(* Logix 5000 project; controller p65 vendor 1 type 14 code 85 rev 20.11; software revision 20.01; part 3 of 7 *)
(* tags used below, declared in another part *)
   BatterycanSupplyPower : ALIAS FOR DINT00_22.0;
   Batterycharge : ALIAS FOR REAL00_3;
   BatteryreqDischarge : ALIAS FOR DINT00_22.30;
   BatteryreqDisconnect : ALIAS FOR DINT00_22.31;
   CommreqConnect : ALIAS FOR DINT00_27.16;
   CommreqDisconnect : ALIAS FOR DINT00_27.17;
   DCMicroGridcanNotifyUser : ALIAS FOR DINT00_23.5;
   DCMicroGridinitialPowerRate : ALIAS FOR REAL00_29;
   DCMicroGridisInOperation : ALIAS FOR DINT00_23.8;
   DCMicroGridisShutdown : ALIAS FOR DINT00_23.9;
   DCMicroGridisSimulating : ALIAS FOR DINT00_23.10;
   DCMicroGridisStarted : ALIAS FOR DINT00_23.11;
   DCMicroGridlowestSupportedPriority : ALIAS FOR DINT00_17;
   DCMicroGridmaxPowerRate : ALIAS FOR REAL00_185;
   DCMicroGridmorePowerAvailable : ALIAS FOR DINT00_32.12;
   DCMicroGridnotificationTimer : ALIAS FOR CLTIMER00_94;
   DCMicroGridpowerRate : ALIAS FOR REAL00_186;
   DCMicroGridpowerRateIncrement : REAL;
   DCMicroGridrecruitingPhase : ALIAS FOR DINT00_18;
   DCMicroGridreqReset : ALIAS FOR DINT00_32.13;
   DCMicroGridreqShutdown : ALIAS FOR DINT00_32.14;
   DCMicroGridreqStartup : ALIAS FOR DINT00_32.15;
   DCMicroGridResetEventFail : ALIAS FOR DINT00_32.16;
   DCMicroGridResetEventSuccess : ALIAS FOR DINT00_32.17;
   DCMicroGridResetFailTimer : ALIAS FOR CLTIMER00_95;
   DCMicroGridResetInProcess : ALIAS FOR DINT00_32.18;
   DCMicroGridResetMsg : ALIAS FOR MESSAGE00_25;
   DCMicroGridResetSuccessTimer : ALIAS FOR CLTIMER00_96;
   DCMicroGridShutdownEventFail : ALIAS FOR DINT00_32.19;
   DCMicroGridShutdownEventSuccess : ALIAS FOR DINT00_32.20;
   DCMicroGridShutdownFailTimer : ALIAS FOR CLTIMER00_97;
   DCMicroGridShutdownInProcess : ALIAS FOR DINT00_32.21;
   DCMicroGridShutdownMsg : ALIAS FOR MESSAGE00_26;
   DCMicroGridShutdownSuccessTimer : ALIAS FOR CLTIMER00_98;
   DCMicroGridsourcesProvidingExcessPower : ALIAS FOR DINT00_33.7;
   DCMicroGridStartupEventFail : ALIAS FOR DINT00_33.8;
   DCMicroGridStartupEventSuccess : ALIAS FOR DINT00_33.9;
   DCMicroGridStartupFailTimer : ALIAS FOR CLTIMER00_100;
   DCMicroGridStartupInProcess : ALIAS FOR DINT00_33.10;
   DCMicroGridStartupMsg : ALIAS FOR MESSAGE00_27;
   DCMicroGridStartupSuccessTimer : ALIAS FOR CLTIMER00_101;
   DCMicroGridtest : ALIAS FOR REAL00_192;
   DCMicroGridtestout : ALIAS FOR REAL00_193;
   DCMicroGriduserNotified : ALIAS FOR DINT00_33.11;
   House01accountBalance : ALIAS FOR REAL00_115;
   House01accountDepositRate : ALIAS FOR REAL00_116;
   House01Bclose : ALIAS FOR Local:3:O.Data.0;
   House01BcloseHILS : ALIAS FOR plc1_local_6[0].0;
   House01BcloseProxy : ALIAS FOR DINT00_28.9;
   House01BintReqClose : ALIAS FOR DINT00_28.10;
   House01BisClosed : ALIAS FOR DINT00_28.11;
   House01BisOpen : ALIAS FOR DINT00_28.12;
   House01BreqClose : ALIAS FOR DINT00_28.13;
   House01BreqOpen : ALIAS FOR DINT00_28.14;
   House01commandChanged : ALIAS FOR DINT00_28.15;
   House01commandChangedTimer : ALIAS FOR CLTIMER00_50;
   House01current : ALIAS FOR REAL00_117;
   House01currentHILS : ALIAS FOR plc1_local_2[0];
   House01currentRaw : ALIAS FOR Local:1:I.Ch12Data;
   House01deadband : ALIAS FOR REAL00_118;
   House01depositTimer : ALIAS FOR CLTIMER00_51;
   House01DisconnectPowerEventFail : ALIAS FOR DINT00_28.16;
   House01DisconnectPowerEventSuccess : ALIAS FOR DINT00_28.17;
   House01DisconnectPowerFailTimer : ALIAS FOR CLTIMER00_52;
   House01DisconnectPowerInProcess : ALIAS FOR DINT00_28.18;
   House01DisconnectPowerMsg : ALIAS FOR MESSAGE00_12;
   House01DisconnectPowerSuccessTimer : ALIAS FOR CLTIMER00_53;
   House01failedToConnect : ALIAS FOR DINT00_28.19;
   House01failedToDisconnect : ALIAS FOR DINT00_28.20;
   House01fundsAvailable : ALIAS FOR DINT00_28.21;
   House01incrementToAdd : ALIAS FOR REAL00_119;
   House01incrementToSubtract : ALIAS FOR REAL00_120;
   House01initialAccountBalance : ALIAS FOR REAL00_121;
   House01intReqConnect : ALIAS FOR DINT00_28.22;
   House01isConnected : ALIAS FOR DINT00_28.23;
   House01isDisconnected : ALIAS FOR DINT00_28.24;
   House01minBalance : ALIAS FOR REAL00_122;
   House01minBalanceToReconnect : ALIAS FOR REAL00_123;
   House01minTime : ALIAS FOR REAL00_124;
   House01powerRate : ALIAS FOR REAL00_125;
   House01powerRateMax : REAL;
   House01priority : ALIAS FOR DINT00_12;
   House01PurchasePowerEventFail : ALIAS FOR DINT00_28.25;
   House01PurchasePowerEventSuccess : ALIAS FOR DINT00_28.26;
   House01PurchasePowerFailTimer : ALIAS FOR CLTIMER00_54;
   House01PurchasePowerInProcess : ALIAS FOR DINT00_28.27;
   House01PurchasePowerMsg : ALIAS FOR MESSAGE00_13;
   House01PurchasePowerSuccessTimer : ALIAS FOR CLTIMER00_55;
   House01reqConnect : ALIAS FOR DINT00_28.28;
   House01reqDisconnect : ALIAS FOR DINT00_28.29;
   House01runningOut : ALIAS FOR DINT00_28.30;
   House01spendingRate : ALIAS FOR REAL00_126;
   House01timeRemaining : ALIAS FOR REAL00_127;
   House01usageTimer : ALIAS FOR CLTIMER00_56;
   House02accountBalance : ALIAS FOR REAL00_128;
   House02initialAccountBalance : ALIAS FOR REAL00_134;
   House02powerRate : ALIAS FOR REAL00_138;
   House02powerRateMax : REAL;
   House02priority : ALIAS FOR DINT00_13;
   House02reqConnect : ALIAS FOR DINT00_29.18;
   House02reqDisconnect : ALIAS FOR DINT00_29.19;
   House03accountBalance : ALIAS FOR REAL00_141;
   House03initialAccountBalance : ALIAS FOR REAL00_147;
   House03powerRate : ALIAS FOR REAL00_151;
   House03powerRateMax : REAL;
   House03priority : ALIAS FOR DINT00_14;
   House03reqConnect : ALIAS FOR DINT00_30.8;
   House03reqDisconnect : ALIAS FOR DINT00_30.9;
   House04accountBalance : ALIAS FOR REAL00_154;
   House04initialAccountBalance : ALIAS FOR REAL00_160;
   House04powerRate : ALIAS FOR REAL00_164;
   House04powerRateMax : REAL;
   House04priority : ALIAS FOR DINT00_15;
   House04reqConnect : ALIAS FOR DINT00_30.30;
   House04reqDisconnect : ALIAS FOR DINT00_30.31;
   House05accountBalance : ALIAS FOR REAL00_167;
   House05initialAccountBalance : ALIAS FOR REAL00_173;
   House05powerRate : ALIAS FOR REAL00_177;
   House05powerRateMax : REAL;
   House05priority : ALIAS FOR DINT00_16;
   House05reqConnect : ALIAS FOR DINT00_31.20;
   House05reqDisconnect : ALIAS FOR DINT00_31.21;
   Load01accountBalance : ALIAS FOR REAL00_37;
   Load01initialAccountBalance : ALIAS FOR REAL00_43;
   Load01powerRate : ALIAS FOR REAL00_47;
   Load01powerRateMax : REAL;
   Load01priority : ALIAS FOR DINT00_5;
   Load01reqConnect : ALIAS FOR DINT00_24.18;
   Load01reqDisconnect : ALIAS FOR DINT00_24.19;
   Load02accountBalance : ALIAS FOR REAL00_50;
   Load02initialAccountBalance : ALIAS FOR REAL00_56;
   Load02powerRate : ALIAS FOR REAL00_60;
   Load02powerRateMax : REAL;
   Load02priority : ALIAS FOR DINT00_6;
   Load02reqConnect : ALIAS FOR DINT00_25.8;
   Load02reqDisconnect : ALIAS FOR DINT00_25.9;
   Load03accountBalance : ALIAS FOR REAL00_63;
   Load03initialAccountBalance : ALIAS FOR REAL00_69;
   Load03powerRate : ALIAS FOR REAL00_73;
   Load03powerRateMax : REAL;
   Load03priority : ALIAS FOR DINT00_7;
   Load03reqConnect : ALIAS FOR DINT00_25.30;
   Load03reqDisconnect : ALIAS FOR DINT00_25.31;
   Load04accountBalance : ALIAS FOR REAL00_76;
   Load04initialAccountBalance : ALIAS FOR REAL00_82;
   Load04powerRate : ALIAS FOR REAL00_86;
   Load04powerRateMax : REAL;
   Load04priority : ALIAS FOR DINT00_8;
   Load04reqConnect : ALIAS FOR DINT00_26.20;
   Load04reqDisconnect : ALIAS FOR DINT00_26.21;
   Load05accountBalance : ALIAS FOR REAL00_89;
   Load05initialAccountBalance : ALIAS FOR REAL00_95;
   Load05powerRate : ALIAS FOR REAL00_99;
   Load05powerRateMax : REAL;
   Load05priority : ALIAS FOR DINT00_9;
   Load05reqConnect : ALIAS FOR DINT00_27.10;
   Load05reqDisconnect : ALIAS FOR DINT00_27.11;
   LoadslowVoltage : ALIAS FOR DINT00_27.23;
   PricedecreaseInProcess : BOOL;
   PriceDecreaseTimer : TIMER;
   PriceIncreaseTimer : TIMER;
   PriorityDecreaseInProcess : BOOL;
   PriorityDecreaseTimer : TIMER;
   PriorityIncreaseTimer : TIMER;
   ResreqConnect : ALIAS FOR DINT00_31.29;
   ResreqDisconnect : ALIAS FOR DINT00_31.30;
   SolarPanelcanSupplyPower : ALIAS FOR DINT00_32.28;
   SolarPanelprovidingExcessPower : ALIAS FOR DINT00_33.4;
   SolarPanelreqConnect : ALIAS FOR DINT00_33.5;
   SolarPanelreqDisconnect : ALIAS FOR DINT00_33.6;
   UsingAgents : BOOL;

PROGRAM DCMicroGrid   (* main routine DCMicroGrid *)

ROUTINE DCMicroGrid   (* ladder *)
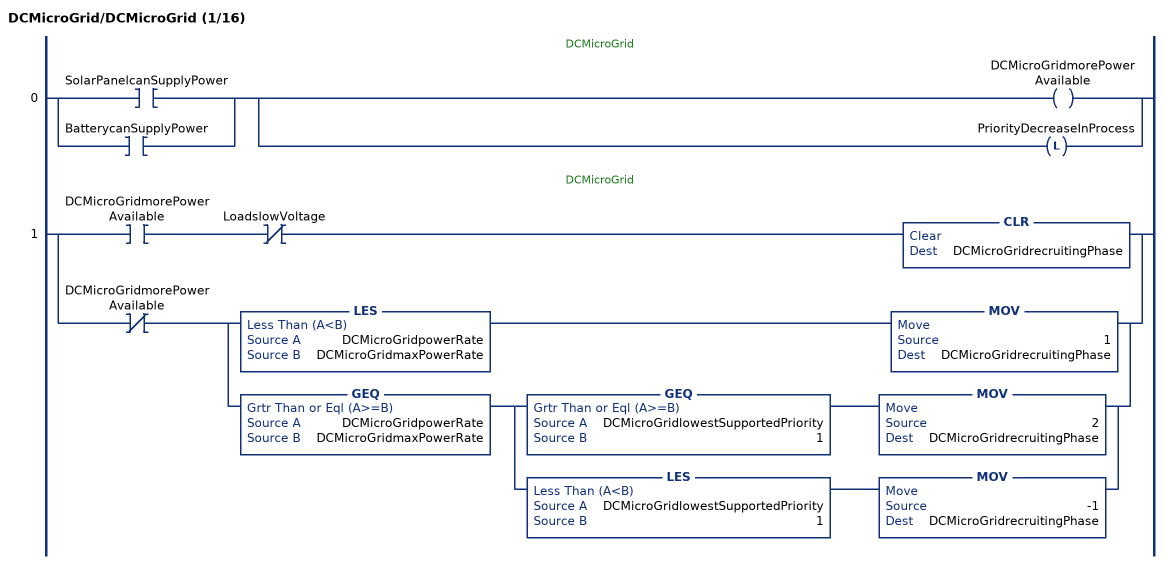
   // DCMicroGrid
   0: [XIC(SolarPanelcanSupplyPower) ,XIC(BatterycanSupplyPower) ][OTE(DCMicroGridmorePowerAvailable) ,OTL(PriorityDecreaseInProcess) ];
   // DCMicroGrid
   1: [XIC(DCMicroGridmorePowerAvailable) XIO(LoadslowVoltage) CLR(DCMicroGridrecruitingPhase) ,XIO(DCMicroGridmorePowerAvailable) [LES(DCMicroGridpowerRate,DCMicroGridmaxPowerRate) MOV(1,DCMicroGridrecruitingPhase) ,GEQ(DCMicroGridpowerRate,DCMicroGridmaxPowerRate) [GEQ(DCMicroGridlowestSupportedPriority,1) MOV(2,DCMicroGridrecruitingPhase) ,LES(DCMicroGridlowestSupportedPriority,1) MOV(-1,DCMicroGridrecruitingPhase) ] ] ];
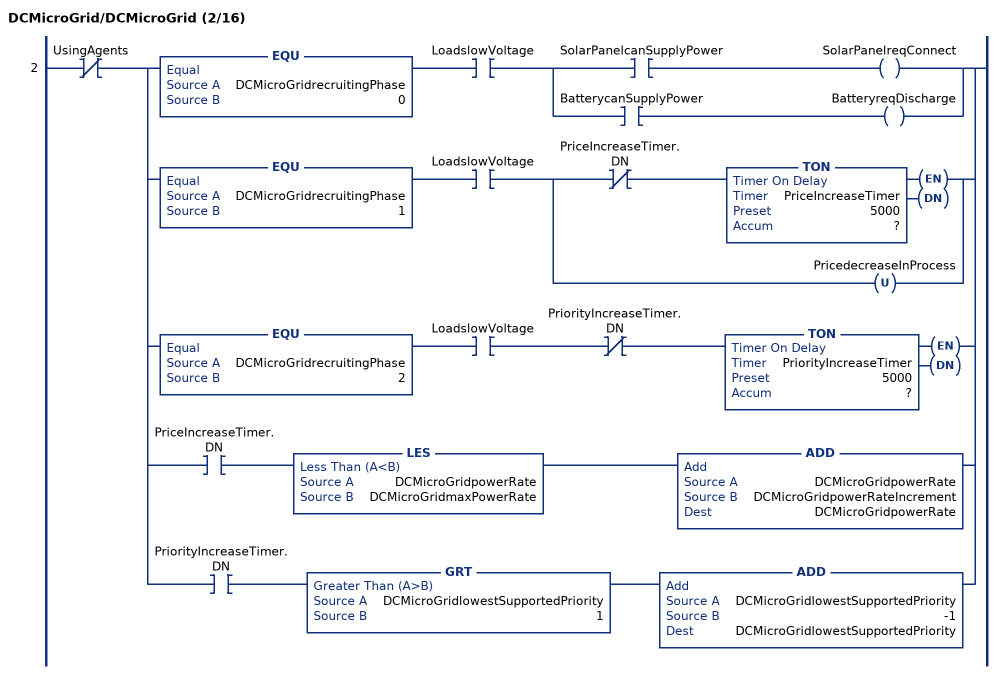
   2: XIO(UsingAgents)[EQU(DCMicroGridrecruitingPhase,0) XIC(LoadslowVoltage) [XIC(SolarPanelcanSupplyPower) OTE(SolarPanelreqConnect) ,XIC(BatterycanSupplyPower) OTE(BatteryreqDischarge) ] ,EQU(DCMicroGridrecruitingPhase,1) XIC(LoadslowVoltage) [XIO(PriceIncreaseTimer.DN) TON(PriceIncreaseTimer,?,?) ,OTU(PricedecreaseInProcess) ] ,EQU(DCMicroGridrecruitingPhase,2) XIC(LoadslowVoltage) XIO(PriorityIncreaseTimer.DN) TON(PriorityIncreaseTimer,?,?) ,XIC(PriceIncreaseTimer.DN) LES(DCMicroGridpowerRate,DCMicroGridmaxPowerRate) ADD(DCMicroGridpowerRate,DCMicroGridpowerRateIncrement,DCMicroGridpowerRate) ,XIC(PriorityIncreaseTimer.DN) GRT(DCMicroGridlowestSupportedPriority,1) ADD(DCMicroGridlowestSupportedPriority,-1,DCMicroGridlowestSupportedPriority) ];
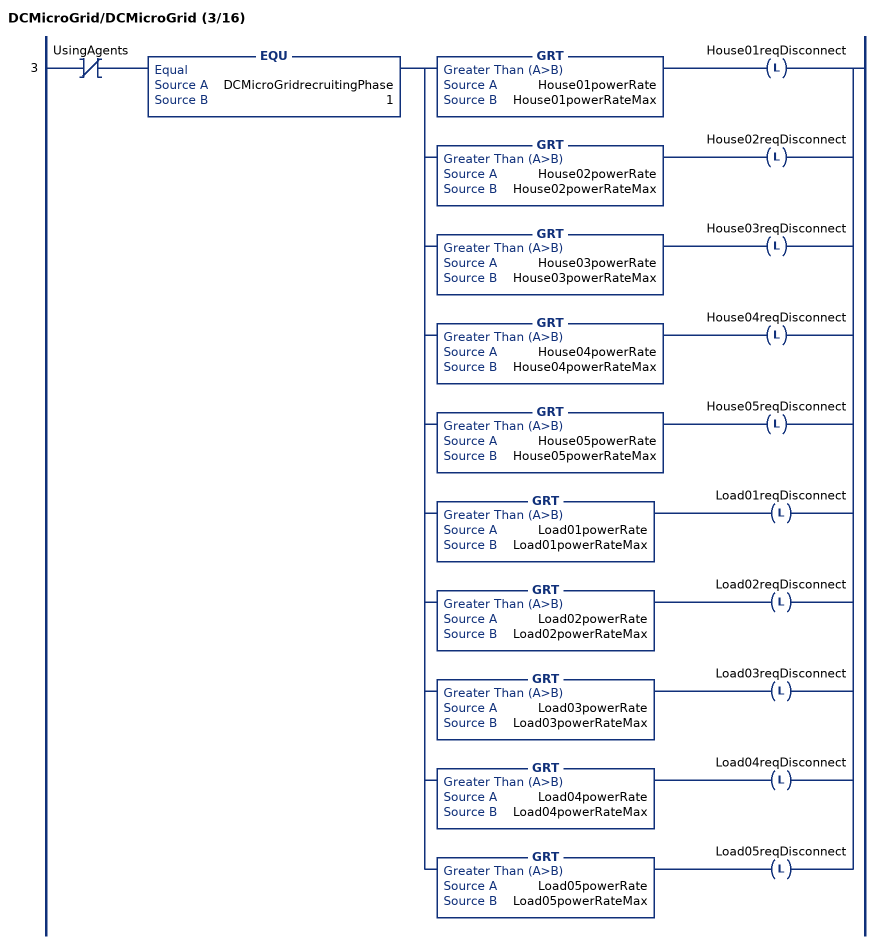
   3: XIO(UsingAgents)EQU(DCMicroGridrecruitingPhase,1)[GRT(House01powerRate,House01powerRateMax) OTL(House01reqDisconnect) ,GRT(House02powerRate,House02powerRateMax) OTL(House02reqDisconnect) ,GRT(House03powerRate,House03powerRateMax) OTL(House03reqDisconnect) ,GRT(House04powerRate,House04powerRateMax) OTL(House04reqDisconnect) ,GRT(House05powerRate,House05powerRateMax) OTL(House05reqDisconnect) ,GRT(Load01powerRate,Load01powerRateMax) OTL(Load01reqDisconnect) ,GRT(Load02powerRate,Load02powerRateMax) OTL(Load02reqDisconnect) ,GRT(Load03powerRate,Load03powerRateMax) OTL(Load03reqDisconnect) ,GRT(Load04powerRate,Load04powerRateMax) OTL(Load04reqDisconnect) ,GRT(Load05powerRate,Load05powerRateMax) OTL(Load05reqDisconnect) ];
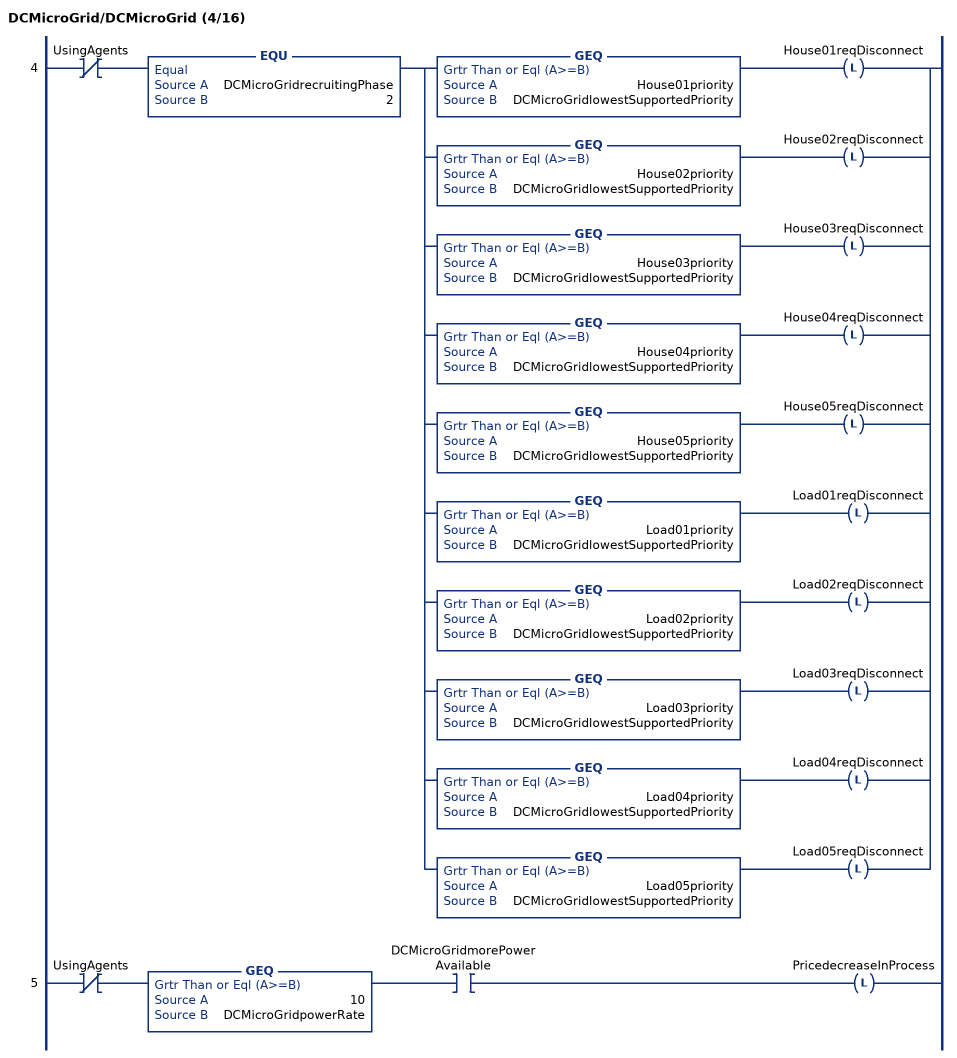
   4: XIO(UsingAgents)EQU(DCMicroGridrecruitingPhase,2)[GEQ(House01priority,DCMicroGridlowestSupportedPriority) OTL(House01reqDisconnect) ,GEQ(House02priority,DCMicroGridlowestSupportedPriority) OTL(House02reqDisconnect) ,GEQ(House03priority,DCMicroGridlowestSupportedPriority) OTL(House03reqDisconnect) ,GEQ(House04priority,DCMicroGridlowestSupportedPriority) OTL(House04reqDisconnect) ,GEQ(House05priority,DCMicroGridlowestSupportedPriority) OTL(House05reqDisconnect) ,GEQ(Load01priority,DCMicroGridlowestSupportedPriority) OTL(Load01reqDisconnect) ,GEQ(Load02priority,DCMicroGridlowestSupportedPriority) OTL(Load02reqDisconnect) ,GEQ(Load03priority,DCMicroGridlowestSupportedPriority) OTL(Load03reqDisconnect) ,GEQ(Load04priority,DCMicroGridlowestSupportedPriority) OTL(Load04reqDisconnect) ,GEQ(Load05priority,DCMicroGridlowestSupportedPriority) OTL(Load05reqDisconnect) ];
   5: XIO(UsingAgents)GEQ(10,DCMicroGridpowerRate)XIC(DCMicroGridmorePowerAvailable)OTL(PricedecreaseInProcess);
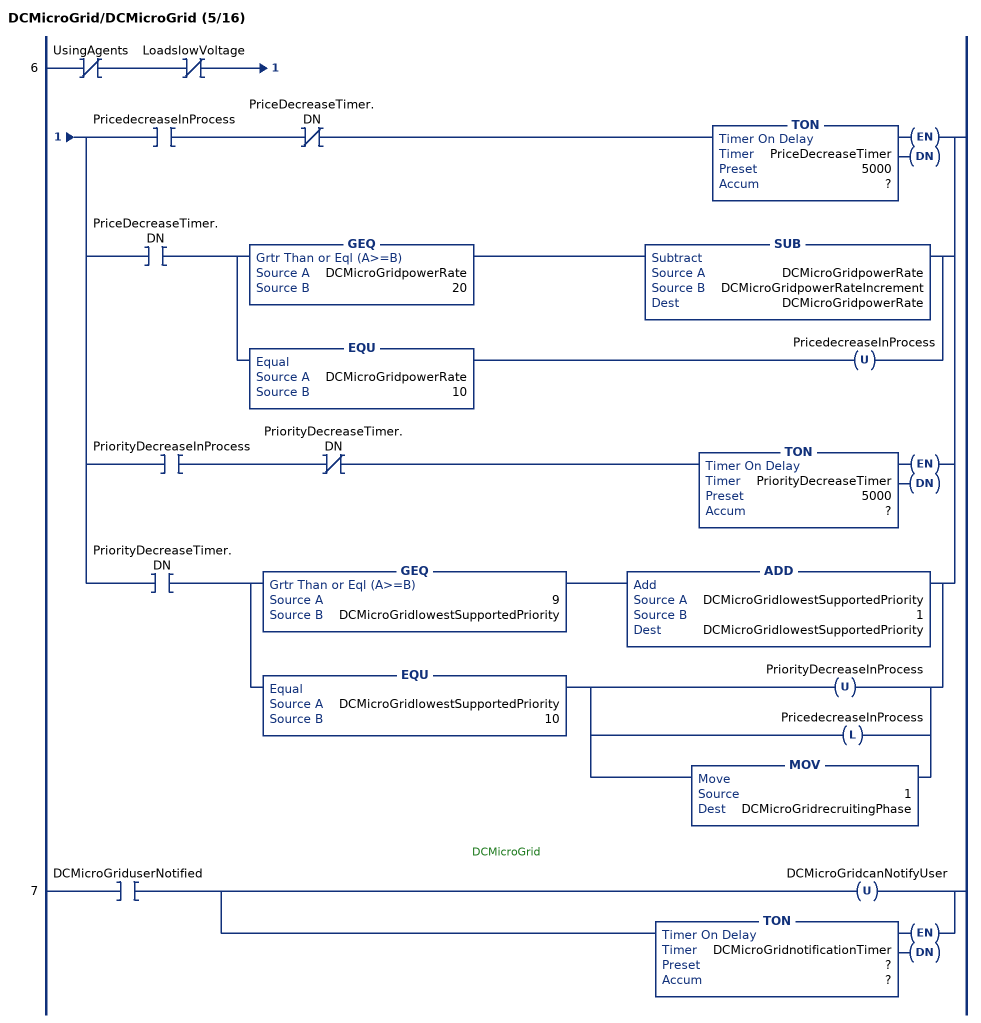
   6: XIO(UsingAgents)XIO(LoadslowVoltage)[XIC(PricedecreaseInProcess) XIO(PriceDecreaseTimer.DN) TON(PriceDecreaseTimer,?,?) ,XIC(PriceDecreaseTimer.DN) [GEQ(DCMicroGridpowerRate,20) SUB(DCMicroGridpowerRate,DCMicroGridpowerRateIncrement,DCMicroGridpowerRate) ,EQU(DCMicroGridpowerRate,10) OTU(PricedecreaseInProcess) ] ,XIC(PriorityDecreaseInProcess) XIO(PriorityDecreaseTimer.DN) TON(PriorityDecreaseTimer,?,?) ,XIC(PriorityDecreaseTimer.DN) [GEQ(9,DCMicroGridlowestSupportedPriority) ADD(DCMicroGridlowestSupportedPriority,1,DCMicroGridlowestSupportedPriority) ,EQU(DCMicroGridlowestSupportedPriority,10) [OTU(PriorityDecreaseInProcess) ,OTL(PricedecreaseInProcess) ,MOV(1,DCMicroGridrecruitingPhase) ] ] ];
   // DCMicroGrid
   7: XIC(DCMicroGriduserNotified)[OTU(DCMicroGridcanNotifyUser) ,TON(DCMicroGridnotificationTimer,?,?) ];
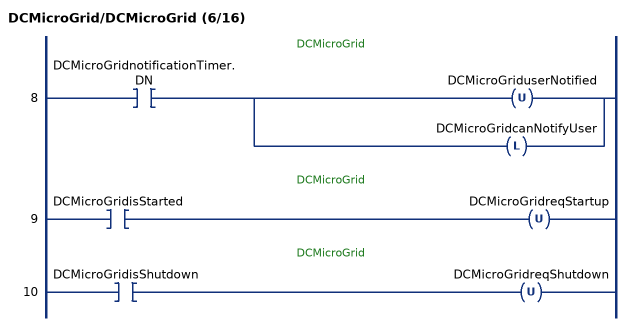
   // DCMicroGrid
   8: XIC(DCMicroGridnotificationTimer.DN)[OTU(DCMicroGriduserNotified) ,OTL(DCMicroGridcanNotifyUser) ];
   // DCMicroGrid
   9: XIC(DCMicroGridisStarted)OTU(DCMicroGridreqStartup);
   // DCMicroGrid
   10: XIC(DCMicroGridisShutdown)OTU(DCMicroGridreqShutdown);
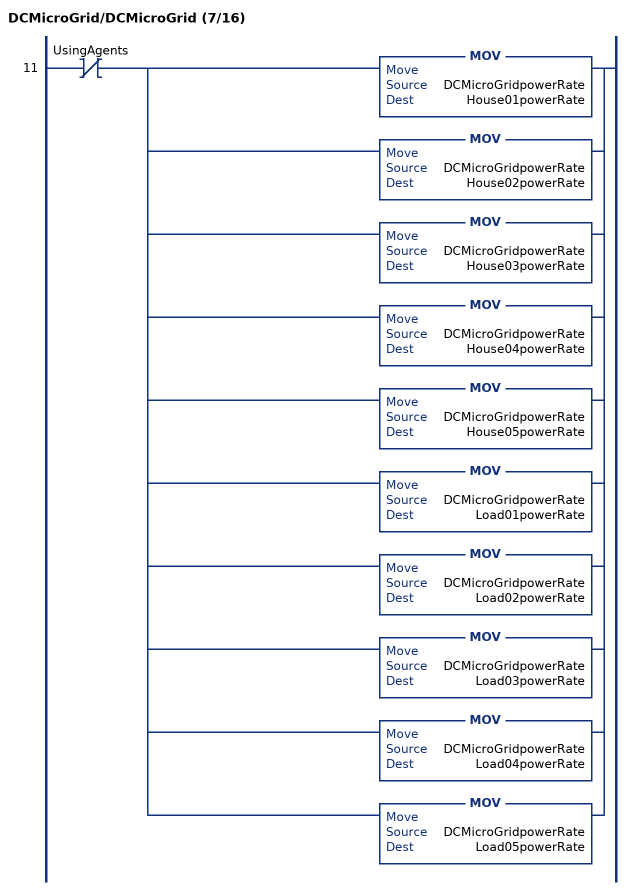
   11: XIO(UsingAgents)[MOV(DCMicroGridpowerRate,House01powerRate) ,MOV(DCMicroGridpowerRate,House02powerRate) ,MOV(DCMicroGridpowerRate,House03powerRate) ,MOV(DCMicroGridpowerRate,House04powerRate) ,MOV(DCMicroGridpowerRate,House05powerRate) ,MOV(DCMicroGridpowerRate,Load01powerRate) ,MOV(DCMicroGridpowerRate,Load02powerRate) ,MOV(DCMicroGridpowerRate,Load03powerRate) ,MOV(DCMicroGridpowerRate,Load04powerRate) ,MOV(DCMicroGridpowerRate,Load05powerRate) ];
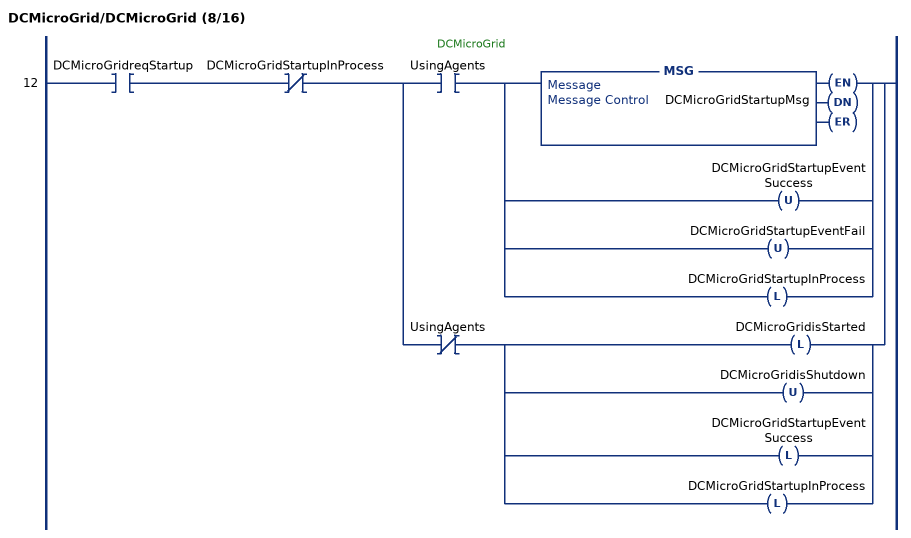
   // DCMicroGrid
   12: XIC(DCMicroGridreqStartup)XIO(DCMicroGridStartupInProcess)[XIC(UsingAgents) [MSG(DCMicroGridStartupMsg) ,OTU(DCMicroGridStartupEventSuccess) ,OTU(DCMicroGridStartupEventFail) ,OTL(DCMicroGridStartupInProcess) ] ,XIO(UsingAgents) [OTL(DCMicroGridisStarted) ,OTU(DCMicroGridisShutdown) ,OTL(DCMicroGridStartupEventSuccess) ,OTL(DCMicroGridStartupInProcess) ] ];
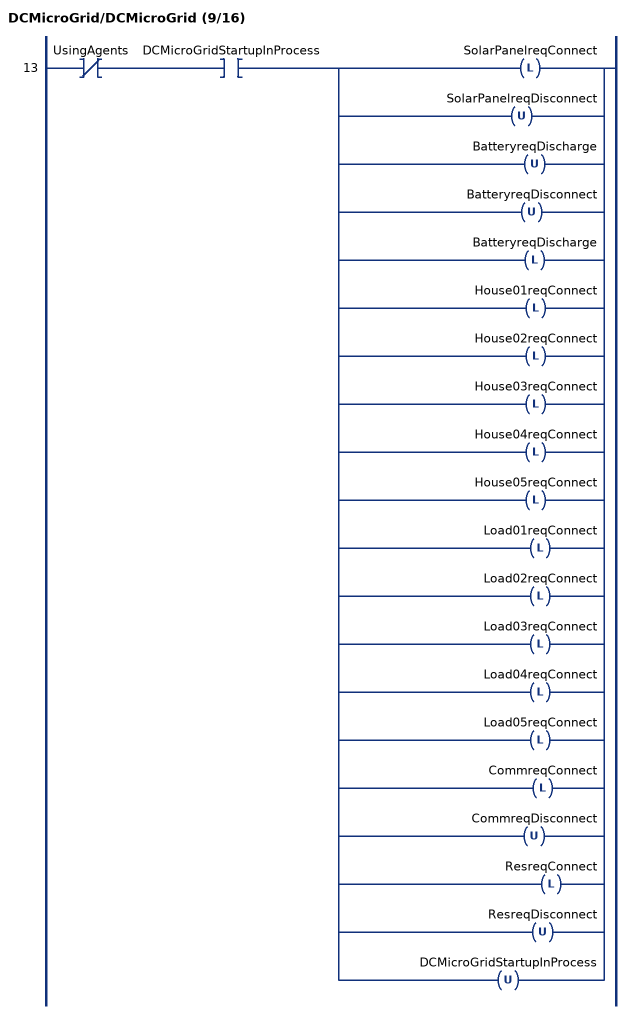
   13: XIO(UsingAgents)XIC(DCMicroGridStartupInProcess)[OTL(SolarPanelreqConnect) ,OTU(SolarPanelreqDisconnect) ,OTU(BatteryreqDischarge) ,OTU(BatteryreqDisconnect) ,OTL(BatteryreqDischarge) ,OTL(House01reqConnect) ,OTL(House02reqConnect) ,OTL(House03reqConnect) ,OTL(House04reqConnect) ,OTL(House05reqConnect) ,OTL(Load01reqConnect) ,OTL(Load02reqConnect) ,OTL(Load03reqConnect) ,OTL(Load04reqConnect) ,OTL(Load05reqConnect) ,OTL(CommreqConnect) ,OTU(CommreqDisconnect) ,OTL(ResreqConnect) ,OTU(ResreqDisconnect) ,OTU(DCMicroGridStartupInProcess) ];
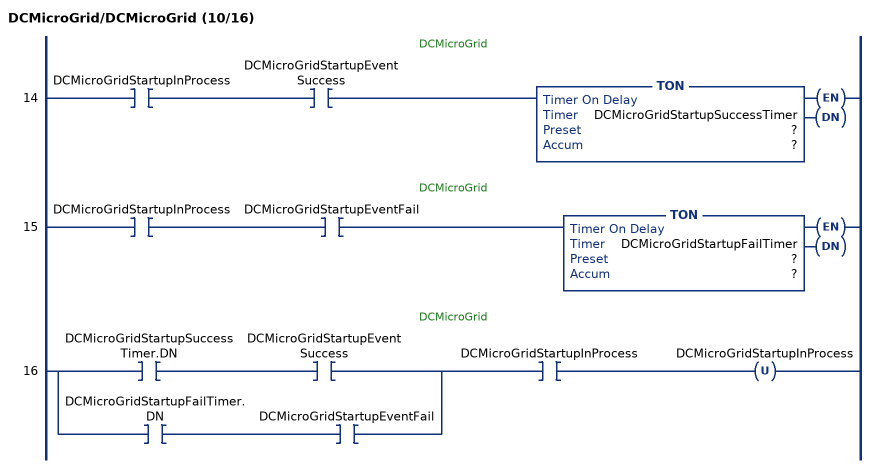
   // DCMicroGrid
   14: XIC(DCMicroGridStartupInProcess)XIC(DCMicroGridStartupEventSuccess)TON(DCMicroGridStartupSuccessTimer,?,?);
   // DCMicroGrid
   15: XIC(DCMicroGridStartupInProcess)XIC(DCMicroGridStartupEventFail)TON(DCMicroGridStartupFailTimer,?,?);
   // DCMicroGrid
   16: [XIC(DCMicroGridStartupSuccessTimer.DN) XIC(DCMicroGridStartupEventSuccess) ,XIC(DCMicroGridStartupFailTimer.DN) XIC(DCMicroGridStartupEventFail) ]XIC(DCMicroGridStartupInProcess)OTU(DCMicroGridStartupInProcess);
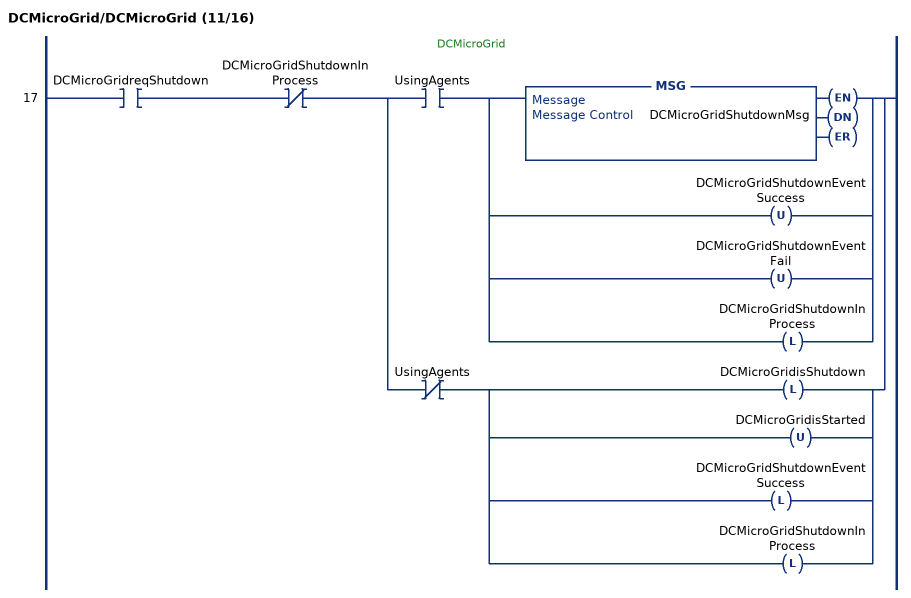
   // DCMicroGrid
   17: XIC(DCMicroGridreqShutdown)XIO(DCMicroGridShutdownInProcess)[XIC(UsingAgents) [MSG(DCMicroGridShutdownMsg) ,OTU(DCMicroGridShutdownEventSuccess) ,OTU(DCMicroGridShutdownEventFail) ,OTL(DCMicroGridShutdownInProcess) ] ,XIO(UsingAgents) [OTL(DCMicroGridisShutdown) ,OTU(DCMicroGridisStarted) ,OTL(DCMicroGridShutdownEventSuccess) ,OTL(DCMicroGridShutdownInProcess) ] ];
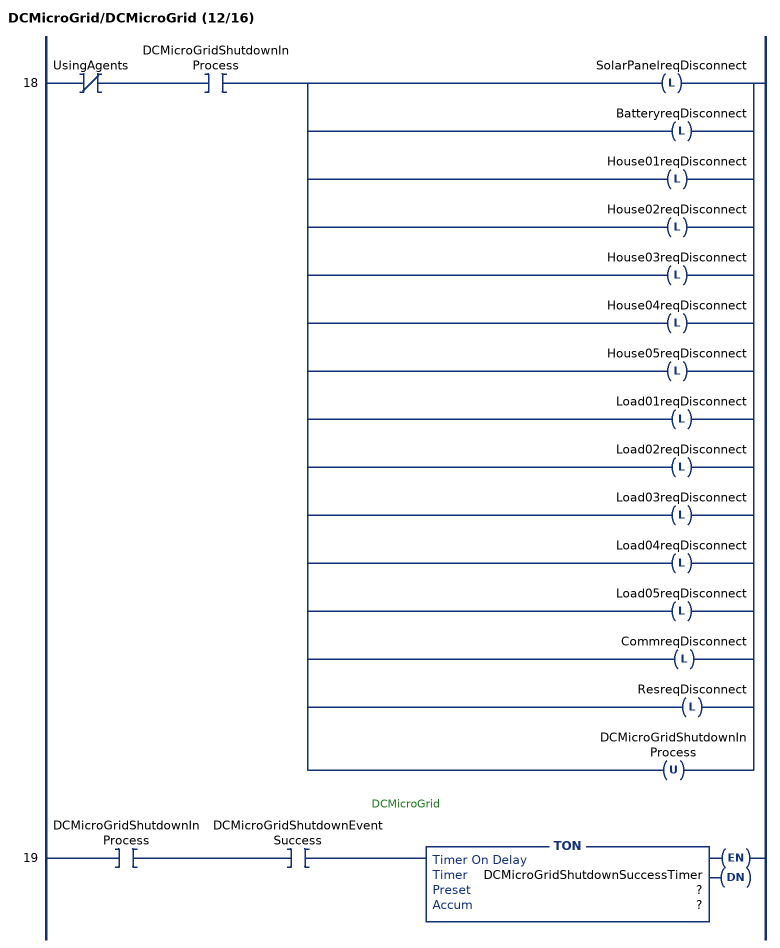
   18: XIO(UsingAgents)XIC(DCMicroGridShutdownInProcess)[OTL(SolarPanelreqDisconnect) ,OTL(BatteryreqDisconnect) ,OTL(House01reqDisconnect) ,OTL(House02reqDisconnect) ,OTL(House03reqDisconnect) ,OTL(House04reqDisconnect) ,OTL(House05reqDisconnect) ,OTL(Load01reqDisconnect) ,OTL(Load02reqDisconnect) ,OTL(Load03reqDisconnect) ,OTL(Load04reqDisconnect) ,OTL(Load05reqDisconnect) ,OTL(CommreqDisconnect) ,OTL(ResreqDisconnect) ,OTU(DCMicroGridShutdownInProcess) ];
   // DCMicroGrid
   19: XIC(DCMicroGridShutdownInProcess)XIC(DCMicroGridShutdownEventSuccess)TON(DCMicroGridShutdownSuccessTimer,?,?);
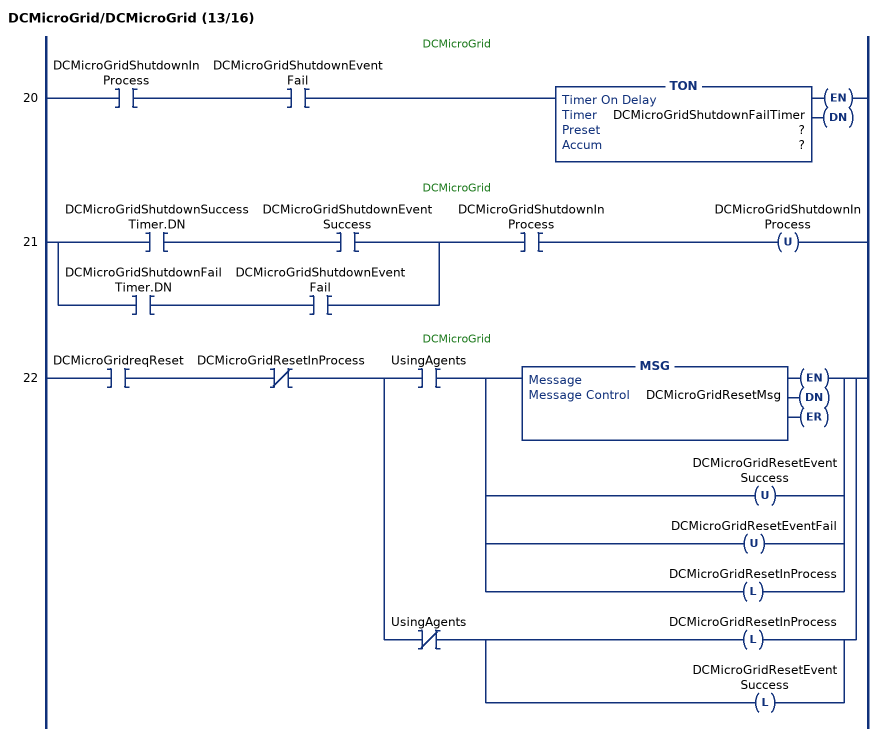
   // DCMicroGrid
   20: XIC(DCMicroGridShutdownInProcess)XIC(DCMicroGridShutdownEventFail)TON(DCMicroGridShutdownFailTimer,?,?);
   // DCMicroGrid
   21: [XIC(DCMicroGridShutdownSuccessTimer.DN) XIC(DCMicroGridShutdownEventSuccess) ,XIC(DCMicroGridShutdownFailTimer.DN) XIC(DCMicroGridShutdownEventFail) ]XIC(DCMicroGridShutdownInProcess)OTU(DCMicroGridShutdownInProcess);
   // DCMicroGrid
   22: XIC(DCMicroGridreqReset)XIO(DCMicroGridResetInProcess)[XIC(UsingAgents) [MSG(DCMicroGridResetMsg) ,OTU(DCMicroGridResetEventSuccess) ,OTU(DCMicroGridResetEventFail) ,OTL(DCMicroGridResetInProcess) ] ,XIO(UsingAgents) [OTL(DCMicroGridResetInProcess) ,OTL(DCMicroGridResetEventSuccess) ] ];
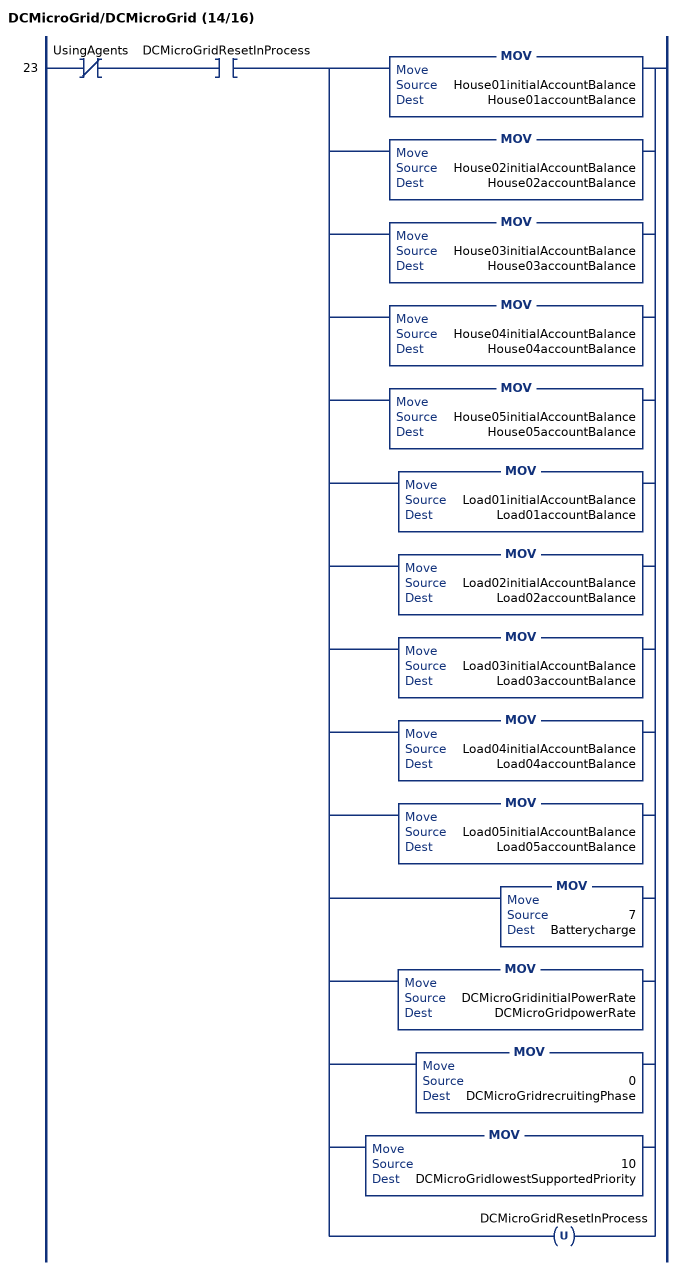
   23: XIO(UsingAgents)XIC(DCMicroGridResetInProcess)[MOV(House01initialAccountBalance,House01accountBalance) ,MOV(House02initialAccountBalance,House02accountBalance) ,MOV(House03initialAccountBalance,House03accountBalance) ,MOV(House04initialAccountBalance,House04accountBalance) ,MOV(House05initialAccountBalance,House05accountBalance) ,MOV(Load01initialAccountBalance,Load01accountBalance) ,MOV(Load02initialAccountBalance,Load02accountBalance) ,MOV(Load03initialAccountBalance,Load03accountBalance) ,MOV(Load04initialAccountBalance,Load04accountBalance) ,MOV(Load05initialAccountBalance,Load05accountBalance) ,MOV(7,Batterycharge) ,MOV(DCMicroGridinitialPowerRate,DCMicroGridpowerRate) ,MOV(0,DCMicroGridrecruitingPhase) ,MOV(10,DCMicroGridlowestSupportedPriority) ,OTU(DCMicroGridResetInProcess) ];
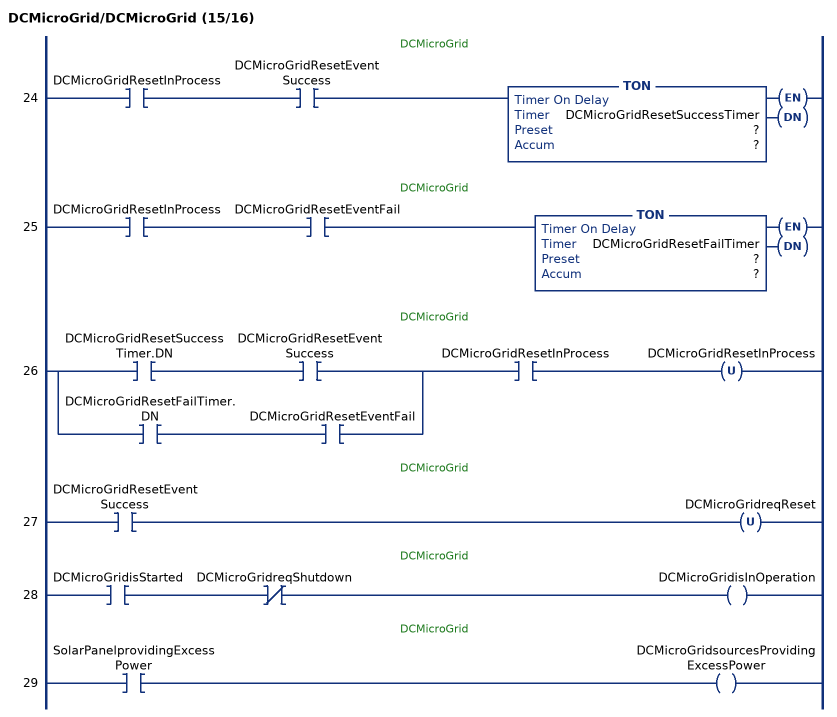
   // DCMicroGrid
   24: XIC(DCMicroGridResetInProcess)XIC(DCMicroGridResetEventSuccess)TON(DCMicroGridResetSuccessTimer,?,?);
   // DCMicroGrid
   25: XIC(DCMicroGridResetInProcess)XIC(DCMicroGridResetEventFail)TON(DCMicroGridResetFailTimer,?,?);
   // DCMicroGrid
   26: [XIC(DCMicroGridResetSuccessTimer.DN) XIC(DCMicroGridResetEventSuccess) ,XIC(DCMicroGridResetFailTimer.DN) XIC(DCMicroGridResetEventFail) ]XIC(DCMicroGridResetInProcess)OTU(DCMicroGridResetInProcess);
   // DCMicroGrid
   27: XIC(DCMicroGridResetEventSuccess)OTU(DCMicroGridreqReset);
   // DCMicroGrid
   28: XIC(DCMicroGridisStarted)XIO(DCMicroGridreqShutdown)OTE(DCMicroGridisInOperation);
   // DCMicroGrid
   29: XIC(SolarPanelprovidingExcessPower)OTE(DCMicroGridsourcesProvidingExcessPower);
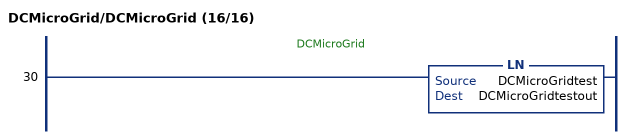
   // DCMicroGrid
   30: LN(DCMicroGridtest,DCMicroGridtestout);
END_ROUTINE
END_PROGRAM

PROGRAM House01   (* main routine House01 *)

ROUTINE House01   (* ladder *)
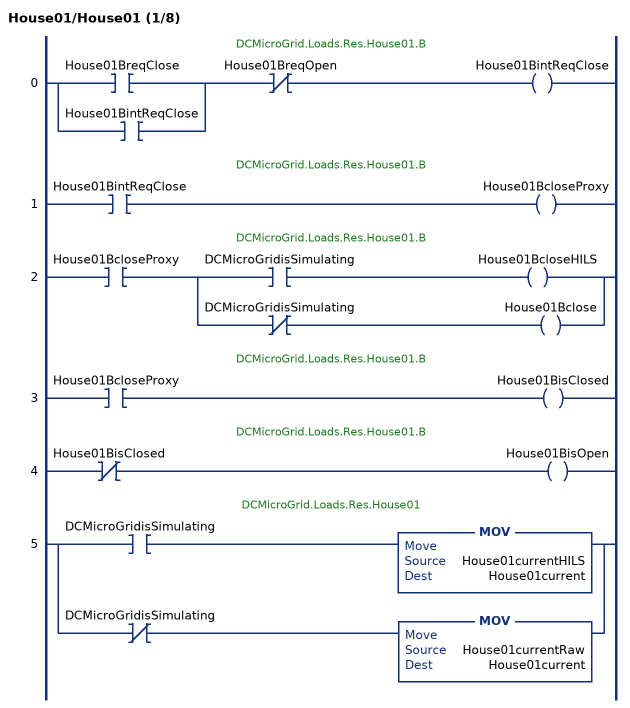
   // DCMicroGrid.Loads.Res.House01.B
   0: [XIC(House01BreqClose) ,XIC(House01BintReqClose) ]XIO(House01BreqOpen)OTE(House01BintReqClose);
   // DCMicroGrid.Loads.Res.House01.B
   1: XIC(House01BintReqClose)OTE(House01BcloseProxy);
   // DCMicroGrid.Loads.Res.House01.B
   2: XIC(House01BcloseProxy)[XIC(DCMicroGridisSimulating) OTE(House01BcloseHILS) ,XIO(DCMicroGridisSimulating) OTE(House01Bclose) ];
   // DCMicroGrid.Loads.Res.House01.B
   3: XIC(House01BcloseProxy)OTE(House01BisClosed);
   // DCMicroGrid.Loads.Res.House01.B
   4: XIO(House01BisClosed)OTE(House01BisOpen);
   // DCMicroGrid.Loads.Res.House01
   5: [XIC(DCMicroGridisSimulating) MOV(House01currentHILS,House01current) ,XIO(DCMicroGridisSimulating) MOV(House01currentRaw,House01current) ];
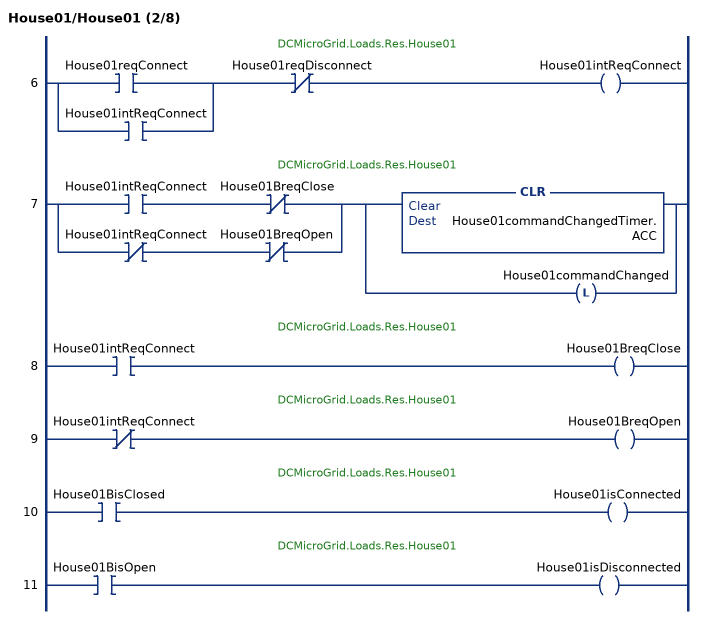
   // DCMicroGrid.Loads.Res.House01
   6: [XIC(House01reqConnect) ,XIC(House01intReqConnect) ]XIO(House01reqDisconnect)OTE(House01intReqConnect);
   // DCMicroGrid.Loads.Res.House01
   7: [XIC(House01intReqConnect) XIO(House01BreqClose) ,XIO(House01intReqConnect) XIO(House01BreqOpen) ][CLR(House01commandChangedTimer.ACC) ,OTL(House01commandChanged) ];
   // DCMicroGrid.Loads.Res.House01
   8: XIC(House01intReqConnect)OTE(House01BreqClose);
   // DCMicroGrid.Loads.Res.House01
   9: XIO(House01intReqConnect)OTE(House01BreqOpen);
   // DCMicroGrid.Loads.Res.House01
   10: XIC(House01BisClosed)OTE(House01isConnected);
   // DCMicroGrid.Loads.Res.House01
   11: XIC(House01BisOpen)OTE(House01isDisconnected);
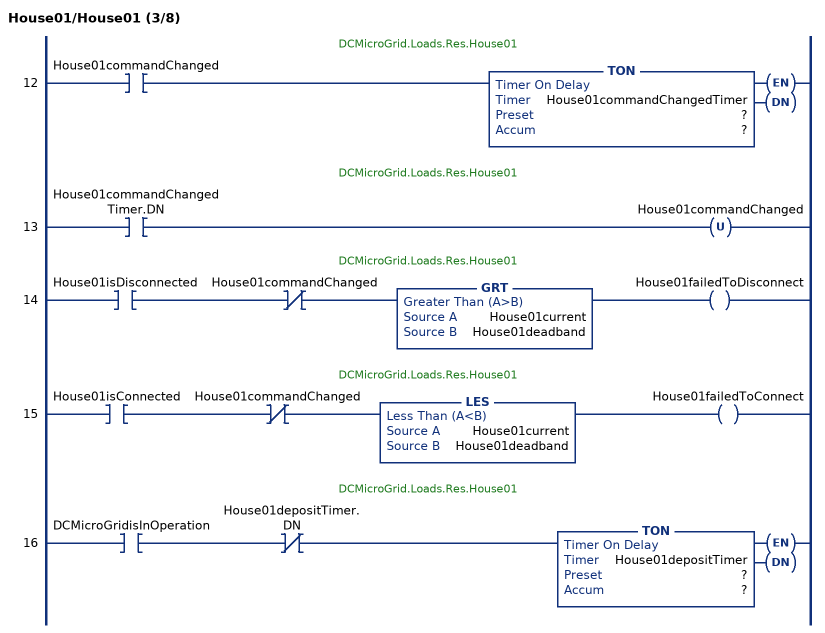
   // DCMicroGrid.Loads.Res.House01
   12: XIC(House01commandChanged)TON(House01commandChangedTimer,?,?);
   // DCMicroGrid.Loads.Res.House01
   13: XIC(House01commandChangedTimer.DN)OTU(House01commandChanged);
   // DCMicroGrid.Loads.Res.House01
   14: XIC(House01isDisconnected)XIO(House01commandChanged)GRT(House01current,House01deadband)OTE(House01failedToDisconnect);
   // DCMicroGrid.Loads.Res.House01
   15: XIC(House01isConnected)XIO(House01commandChanged)LES(House01current,House01deadband)OTE(House01failedToConnect);
   // DCMicroGrid.Loads.Res.House01
   16: XIC(DCMicroGridisInOperation)XIO(House01depositTimer.DN)TON(House01depositTimer,?,?);
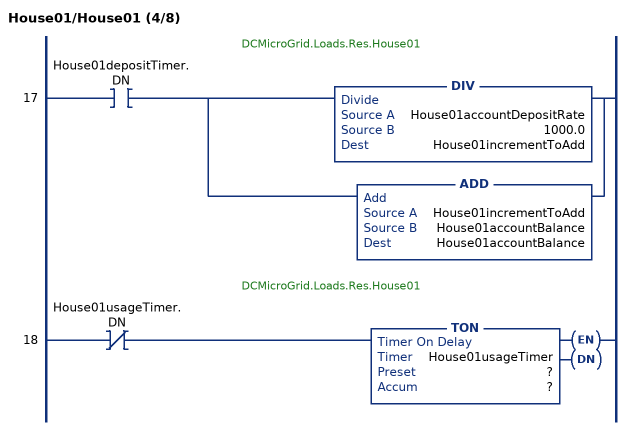
   // DCMicroGrid.Loads.Res.House01
   17: XIC(House01depositTimer.DN)[DIV(House01accountDepositRate,1000.0,House01incrementToAdd) ,ADD(House01incrementToAdd,House01accountBalance,House01accountBalance) ];
   // DCMicroGrid.Loads.Res.House01
   18: XIO(House01usageTimer.DN)TON(House01usageTimer,?,?);
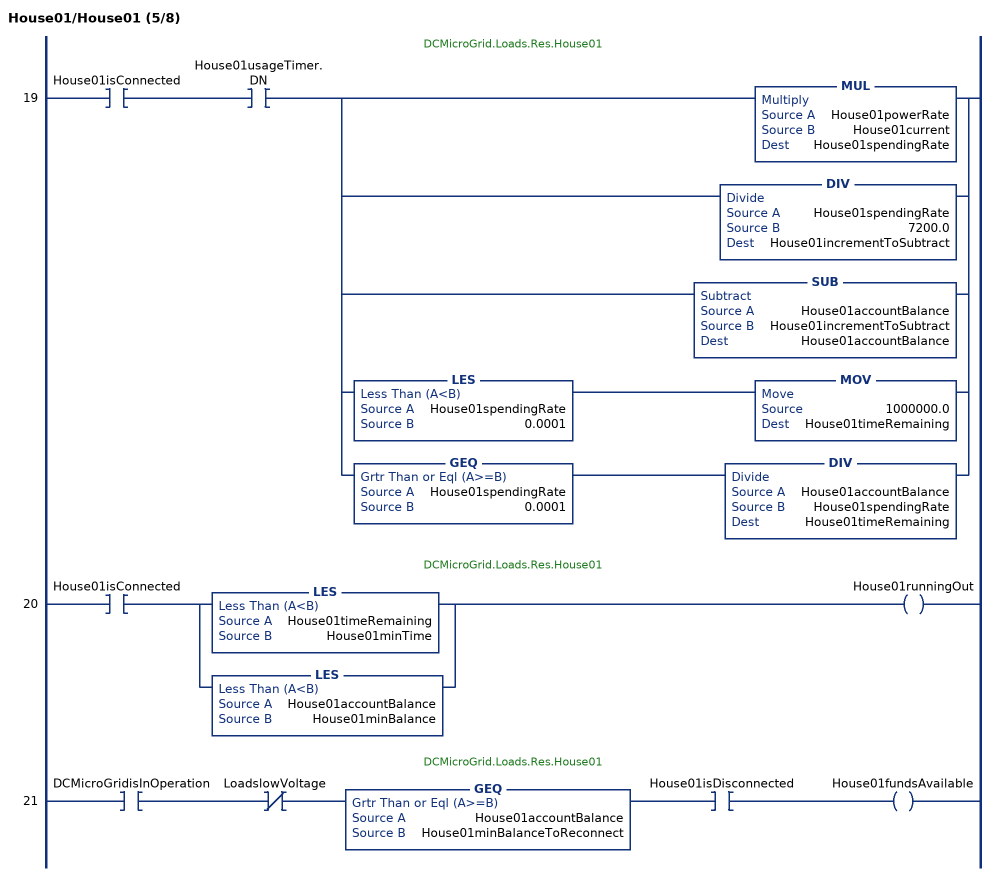
   // DCMicroGrid.Loads.Res.House01
   19: XIC(House01isConnected)XIC(House01usageTimer.DN)[MUL(House01powerRate,House01current,House01spendingRate) ,DIV(House01spendingRate,7200.0,House01incrementToSubtract) ,SUB(House01accountBalance,House01incrementToSubtract,House01accountBalance) ,[LES(House01spendingRate,0.0001) MOV(1000000.0,House01timeRemaining) ,GEQ(House01spendingRate,0.0001) DIV(House01accountBalance,House01spendingRate,House01timeRemaining) ] ];
   // DCMicroGrid.Loads.Res.House01
   20: XIC(House01isConnected)[LES(House01timeRemaining,House01minTime) ,LES(House01accountBalance,House01minBalance) ]OTE(House01runningOut);
   // DCMicroGrid.Loads.Res.House01
   21: XIC(DCMicroGridisInOperation)XIO(LoadslowVoltage)GEQ(House01accountBalance,House01minBalanceToReconnect)XIC(House01isDisconnected)OTE(House01fundsAvailable);
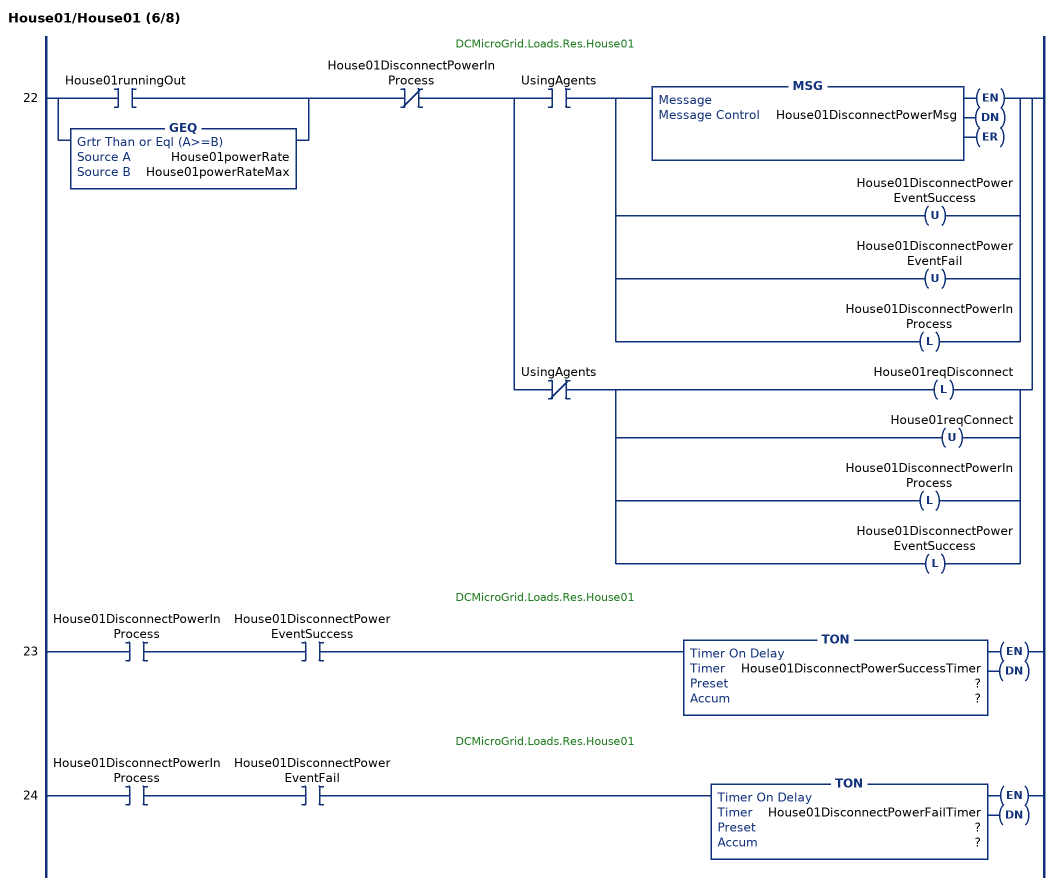
   // DCMicroGrid.Loads.Res.House01
   22: [XIC(House01runningOut) ,GEQ(House01powerRate,House01powerRateMax) ]XIO(House01DisconnectPowerInProcess)[XIC(UsingAgents) [MSG(House01DisconnectPowerMsg) ,OTU(House01DisconnectPowerEventSuccess) ,OTU(House01DisconnectPowerEventFail) ,OTL(House01DisconnectPowerInProcess) ] ,XIO(UsingAgents) [OTL(House01reqDisconnect) ,OTU(House01reqConnect) ,OTL(House01DisconnectPowerInProcess) ,OTL(House01DisconnectPowerEventSuccess) ] ];
   // DCMicroGrid.Loads.Res.House01
   23: XIC(House01DisconnectPowerInProcess)XIC(House01DisconnectPowerEventSuccess)TON(House01DisconnectPowerSuccessTimer,?,?);
   // DCMicroGrid.Loads.Res.House01
   24: XIC(House01DisconnectPowerInProcess)XIC(House01DisconnectPowerEventFail)TON(House01DisconnectPowerFailTimer,?,?);
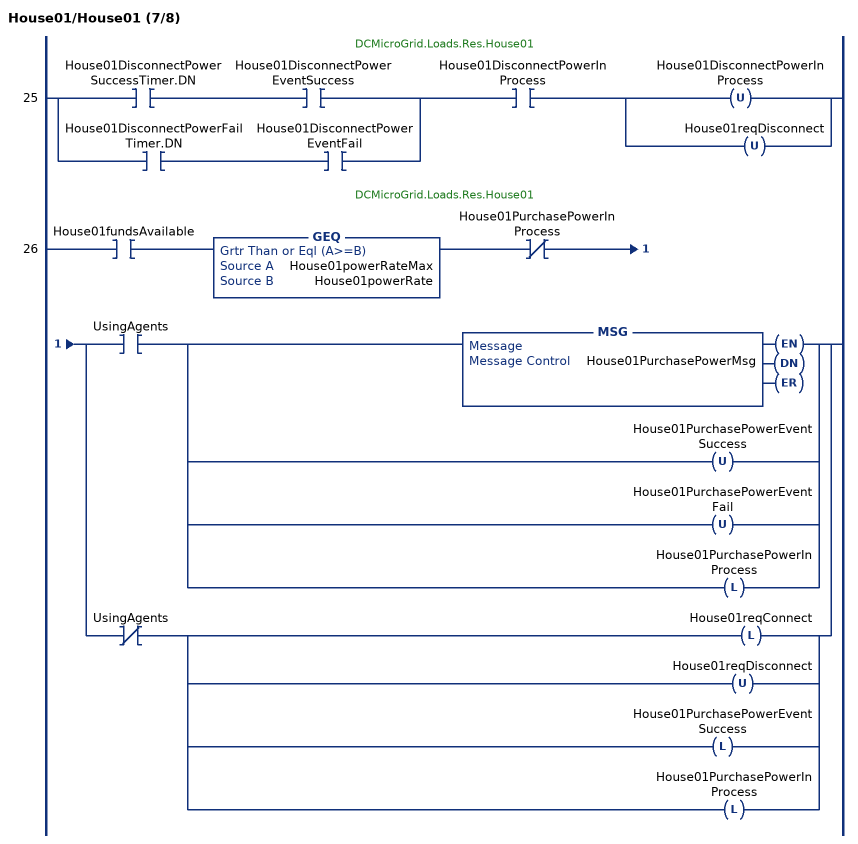
   // DCMicroGrid.Loads.Res.House01
   25: [XIC(House01DisconnectPowerSuccessTimer.DN) XIC(House01DisconnectPowerEventSuccess) ,XIC(House01DisconnectPowerFailTimer.DN) XIC(House01DisconnectPowerEventFail) ]XIC(House01DisconnectPowerInProcess)[OTU(House01DisconnectPowerInProcess) ,OTU(House01reqDisconnect) ];
   // DCMicroGrid.Loads.Res.House01
   26: XIC(House01fundsAvailable)GEQ(House01powerRateMax,House01powerRate)XIO(House01PurchasePowerInProcess)[XIC(UsingAgents) [MSG(House01PurchasePowerMsg) ,OTU(House01PurchasePowerEventSuccess) ,OTU(House01PurchasePowerEventFail) ,OTL(House01PurchasePowerInProcess) ] ,XIO(UsingAgents) [OTL(House01reqConnect) ,OTU(House01reqDisconnect) ,OTL(House01PurchasePowerEventSuccess) ,OTL(House01PurchasePowerInProcess) ] ];
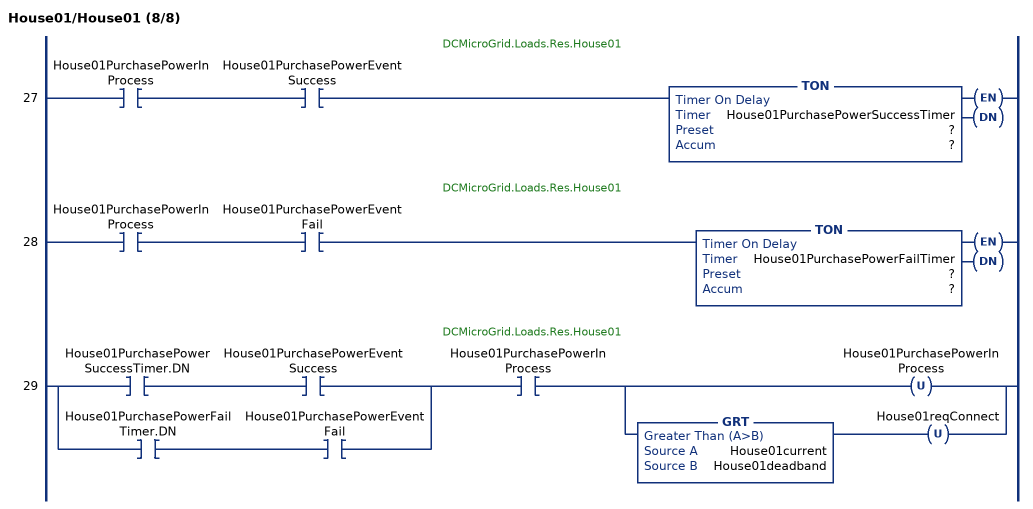
   // DCMicroGrid.Loads.Res.House01
   27: XIC(House01PurchasePowerInProcess)XIC(House01PurchasePowerEventSuccess)TON(House01PurchasePowerSuccessTimer,?,?);
   // DCMicroGrid.Loads.Res.House01
   28: XIC(House01PurchasePowerInProcess)XIC(House01PurchasePowerEventFail)TON(House01PurchasePowerFailTimer,?,?);
   // DCMicroGrid.Loads.Res.House01
   29: [XIC(House01PurchasePowerSuccessTimer.DN) XIC(House01PurchasePowerEventSuccess) ,XIC(House01PurchasePowerFailTimer.DN) XIC(House01PurchasePowerEventFail) ]XIC(House01PurchasePowerInProcess)[OTU(House01PurchasePowerInProcess) ,GRT(House01current,House01deadband) OTU(House01reqConnect) ];
END_ROUTINE
END_PROGRAM
